// TIA Portal V19 export
FUNCTION_BLOCK "Calculator"   // FB10, LAD
{ S7_Optimized_Access := 'TRUE' }
// stored: AutoNumber false, MemoryReserve 100, SetENOAutomatically false
   VAR_INPUT
      value1 : Int;
      value2 : Int;
      add : Bool;
      subtract : Bool;
      multiply : Bool;
      divide : Bool;
   END_VAR
   VAR_OUTPUT
      result : Int;
   END_VAR
BEGIN

REGION Network 1: Add
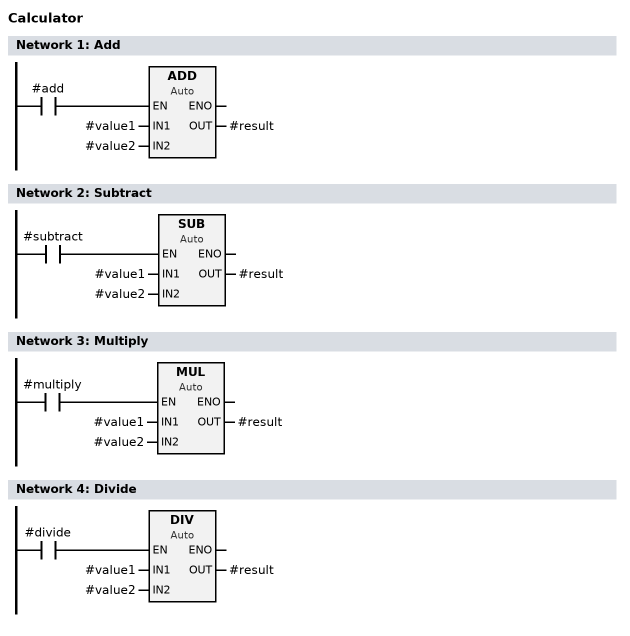
   RUNG wire#powerrail
      Contact( #add )
      Add(in1 := #value1, in2 := #value2, out => #result)
   END_RUNG
   // the same network as SCL:
   IF #add THEN #result := #value1 + #value2; END_IF;
END_REGION

REGION Network 2: Subtract
   RUNG wire#powerrail
      Contact( #subtract )
      Sub(in1 := #value1, in2 := #value2, out => #result)
   END_RUNG
   // the same network as SCL:
   IF #subtract THEN #result := #value1 - #value2; END_IF;
END_REGION

REGION Network 3: Multiply
   RUNG wire#powerrail
      Contact( #multiply )
      Mul(in1 := #value1, in2 := #value2, out => #result)
   END_RUNG
   // the same network as SCL:
   IF #multiply THEN #result := #value1 * #value2; END_IF;
END_REGION

REGION Network 4: Divide
   RUNG wire#powerrail
      Contact( #divide )
      Div(in1 := #value1, in2 := #value2, out => #result)
   END_RUNG
   // the same network as SCL:
   IF #divide THEN #result := #value1 / #value2; END_IF;
END_REGION
END_FUNCTION_BLOCK
